// TIA Portal V19 export
DATA_BLOCK "AUTO P_TRIG"   // DB71
{ S7_Optimized_Access := 'TRUE' }
// stored: MemoryReserve 100
   VAR
      "1" : Bool;
      "2" : Bool;
      "3" : Bool;
      "4" : Bool;
      "5" : Bool;
      "6" : Bool;
      "7" : Bool;
      "8" : Bool;
      "9" : Bool;
      "10" : Bool;
      "11" : Bool;
      "12" : Bool;
      "13" : Bool;
      "14" : Bool;
      "15" : Bool;
      "16" : Bool;
      "17" : Bool;
      "18" : Bool;
      "19" : Bool;
      "20" : Bool;
      "21" : Bool;
      "22" : Bool;
      "23" : Bool;
      "24" : Bool;
      "25" : Bool;
      "26" : Bool;
      "27" : Bool;
      "28" : Bool;
      "29" : Bool;
      "30" : Bool;
   END_VAR
BEGIN
END_DATA_BLOCK
